// TIA Portal V20 export
// export: Created 2025-12-01T14:57:17.1875181Z, ExportSetting None, DisplayName Totally Integrated Automation Portal, DisplayVersion V20 Update 3, DisplayName TIA Portal Openness, DisplayVersion V20 Update 3, DisplayName TIA Portal Version Control Interface, DisplayVersion V20 Update 3, DisplayName STEP 7 Professional, DisplayVersion V20 Update 3, DisplayName STEP 7 Safety, DisplayVersion V20 Update 2, DisplayName WinCC Basic/Comfort/Advanced, DisplayVersion V20 Update 3, DisplayName WinCC Professional, DisplayVersion V20 Update 3, DisplayName WinCC Unified, DisplayVersion V20 Update 3
DATA_BLOCK "DB932_Datos_VarLENZE"   // DB932
{ S7_Optimized_Access := 'FALSE' }
AUTHOR : LENZE
NAME : 20130301
VERSION : 3.0
// stored: AutoNumber false
   VAR
      Red_01 { S7_SetPoint := 'True'} : Array[1..255] of "UDT_VarLenze";   // Red 01 de Variadores Lenze
      Red_02 { S7_SetPoint := 'True'} : Array[1..255] of "UDT_VarLenze";   // Red 02 de Variadores Lenze
   END_VAR
BEGIN
END_DATA_BLOCK
